FUNCTION_BLOCK TimerServer_Delay_backup (* Updates time upon every REQ event and can be used to request time remotely. *)
  (* Standard: 61499-2 *)
  (* Version 1.0, 2017-09-05, Marc Jakobi, HTW Berlin *)
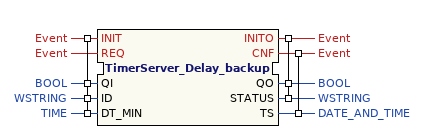
  EVENT_INPUT
    INIT WITH QI, ID, DT_MIN; (* Initialization Request *)
    REQ; (* Service Request Event *)
  END_EVENT
  EVENT_OUTPUT
    INITO WITH QO, STATUS; (* Initialization Confirm *)
    CNF WITH TS; (* Service Indication *)
  END_EVENT
  VAR_INPUT
    QI : BOOL; (* Input event qualifier *)
    ID : WSTRING; (* Connection identifier *)
    DT_MIN : TIME;
  END_VAR
  VAR_OUTPUT
    QO : BOOL; (* Output event qualifier *)
    STATUS : WSTRING; (* Service status *)
    TS : DATE_AND_TIME; (* Time stamp *)
  END_VAR
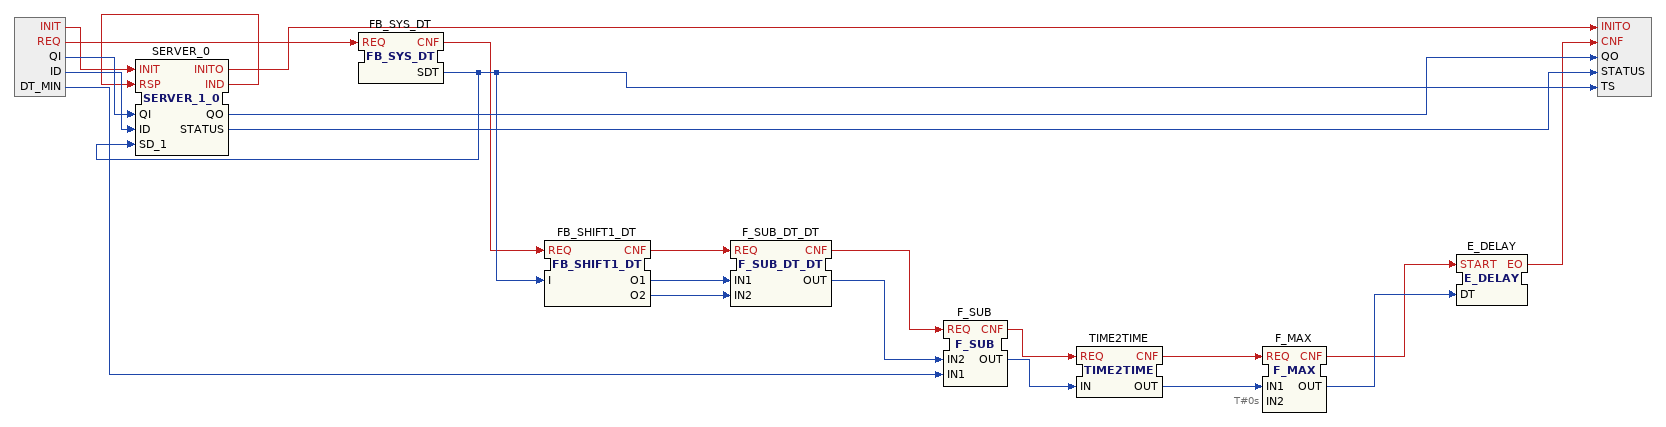
  FBS
    FB_SYS_DT : FB_SYS_DT;
    SERVER_0 : SERVER_1_0;
    FB_SHIFT1_DT : FB_SHIFT1_DT;
    F_SUB_DT_DT : F_SUB_DT_DT;
    F_SUB : F_SUB;
    F_MAX : F_MAX(IN2 := T#0s);
    TIME2TIME : TIME2TIME;
    E_DELAY : E_DELAY;
  END_FBS
  EVENT_CONNECTIONS
    INIT TO SERVER_0.INIT;
    SERVER_0.INITO TO INITO;
    REQ TO FB_SYS_DT.REQ;
    SERVER_0.IND TO SERVER_0.RSP;
    FB_SHIFT1_DT.CNF TO F_SUB_DT_DT.REQ;
    F_SUB_DT_DT.CNF TO F_SUB.REQ;
    FB_SYS_DT.CNF TO FB_SHIFT1_DT.REQ;
    F_SUB.CNF TO TIME2TIME.REQ;
    TIME2TIME.CNF TO F_MAX.REQ;
    F_MAX.CNF TO E_DELAY.START;
    E_DELAY.EO TO CNF;
  END_CONNECTIONS
  DATA_CONNECTIONS
    FB_SYS_DT.SDT TO TS;
    QI TO SERVER_0.QI;
    ID TO SERVER_0.ID;
    SERVER_0.QO TO QO;
    SERVER_0.STATUS TO STATUS;
    FB_SYS_DT.SDT TO SERVER_0.SD_1;
    FB_SYS_DT.SDT TO FB_SHIFT1_DT.I;
    FB_SHIFT1_DT.O1 TO F_SUB_DT_DT.IN1;
    FB_SHIFT1_DT.O2 TO F_SUB_DT_DT.IN2;
    F_SUB_DT_DT.OUT TO F_SUB.IN2;
    DT_MIN TO F_SUB.IN1;
    F_SUB.OUT TO TIME2TIME.IN;
    TIME2TIME.OUT TO F_MAX.IN1;
    F_MAX.OUT TO E_DELAY.DT;
  END_CONNECTIONS
END_FUNCTION_BLOCK
